Staubli VAL3: Form_PanelList.pgx

public program Form_PanelList(string x_sTitle, string x_sPanelTitle, string& x_sList[], num& x_nSelectIndex, string x_sBottom)
begin

//cls()
title(x_sTitle)
call Control_LeftS(x_sBottom)
call Control_PanelS(x_sPanelTitle,22,0,15,10)
call Control_BottomS(x_sBottom)
call Control_List(x_sList,x_nSelectIndex)



end
